(* CODESYS project DiagnosisEtherCAT.library
   Author: TK
   Version: 0.0.9.1
   Description: EtherCATのマスター、スレーブの診断用FBのライブラリです。
   Title: Tk_Diagnosis_EtherCAT
   Placeholder: Tk_Diagnosis_EtherCAT
   Company: Komatsu

Project tree, tasks and I/O mapping:
  libraries: Tc2_Standard, * (Beckhoff Automation GmbH); Tc2_System, * (Beckhoff Automation GmbH); Tc3_EventLogger, * (Beckhoff Automation GmbH)
  EtherCAT Master/
    Base/
      function block FB_DevStateDiagnosis [ST]: FB_Init
      function block FB_FrmStateDiagnosis [ST]: FB_Init
      function block FB_FrmWcStateDiagnosis [ST]: FB_Init
      function block FB_SlaveCountDiagnosis [ST]: FB_Init
    function block FB_DiagnosisEtherCATMaster [ST]
  EtherCAT Slave/
    Base/
      function block FB_StateDiagnosis [ST]: FB_Init
      function block FB_WcStateDiagnosis [ST]: FB_Init
    function block FB_DiagnosisEtherCATSlaveWc0 [ST]: bError, Execute
    function block FB_DiagnosisEtherCATSlaveWc1 [ST]: bError, Execute
    function block FB_DiagnosisEtherCATSlaveWc2 [ST]: bError, Execute
    interface I_DiagnosisEtherCATSlave: bError, Execute
  Example FB/
    function block FB_DiagnosisEtherCATExample [ST]: EtherCATMasterDiagnosis, EtherCATSlaveDiagnosis
  Version/
    global variables Global_Version
*)

// Version/Global_Version
{attribute 'TcGenerated'}
{attribute 'no-analysis'}
{attribute 'linkalways'}
// This function has been automatically generated from the project information.
VAR_GLOBAL CONSTANT
	{attribute 'const_non_replaced'}
	stLibVersion_Tk_Diagnosis_EtherCAT : ST_LibVersion := (iMajor := 0, iMinor := 0, iBuild := 9, iRevision := 1, nFlags := 0, sVersion := '0.0.9.1');
END_VAR

// EtherCAT Master/Base/FB_DevStateDiagnosis
FUNCTION_BLOCK FB_DevStateDiagnosis
VAR CONSTANT
	uiFaultMask					:UINT	:=2#0001_1111_1111_0011;	//デバイスエラーのマスク
END_VAR
VAR_INPUT
	sMasterName					:STRING	:='NameNotSet';				//マスター名
END_VAR
VAR_OUTPUT
	bError						:BOOL;								//エラー発生を出力
END_VAR
VAR
	uiDevState 			AT%I*	:UINT;								//PDデータとリンク
		
	bErrorState					:ARRAY[0..15] OF BOOL;				//各ステートエラー
	fbBitREdge					:ARRAY[0..15] OF R_TRIG;
	fbMessage					:ARRAY[0..15] OF FB_TcMessage;
	i							:INT;
END_VAR

//エラー状態を出力
	bError:= (uiDevState AND uiFaultMask)<>0 ;

//デバイスの状態チェック、エラーは複数発生する可能性があるので全bitチェック
	FOR i := 0 TO 15 DO
		bErrorState[i]:=(uiDevState AND SHL(1,i))<>0;
	END_FOR

//結果をEventloggerへ
	FOR i := 0 TO 15 BY 1 DO
		fbBitREdge[i](CLK:=bErrorState[i]);
		
		IF fbBitREdge[i].Q THEN
			fbMessage[i].ipArguments.Clear().AddString(sMasterName);
			fbMessage[i].Send();
		END_IF
		
	END_FOR

//FB_Init は常に暗黙的に使用可能で、主に初期化に使用されます。
//戻り値は評価されません。特定の結果を得るために、メソッドを明示的に宣言し、
//そのメソッドに標準の初期化コードをもったコードを追加することができます。戻り値を評価できます。
METHOD FB_Init: BOOL
VAR_INPUT
    bInitRetains: BOOL; // TRUE: 保持変数は初期化されます (ウォーム リセット、あるいはコールド リセット)
    bInCopyCode: BOOL;  // TRUE: 後でコードをコピーする (オンライン変更) ために、インスタンスをコピーします。
END_VAR
fbMessage[0].CreateEx(TC_EVENTS.TkEtherCATMasterDiagnosisEventClass.LinkError);
fbMessage[1].CreateEx(TC_EVENTS.TkEtherCATMasterDiagnosisEventClass.IOLockedAfterLinkErrorIOResetRequired);
fbMessage[2].CreateEx(TC_EVENTS.TkEtherCATMasterDiagnosisEventClass.LinkErrorRedundancyAdapter);
fbMessage[3].CreateEx(TC_EVENTS.TkEtherCATMasterDiagnosisEventClass.MissingOneFrameRedundancyAdapter);
fbMessage[4].CreateEx(TC_EVENTS.TkEtherCATMasterDiagnosisEventClass.OutOfSendResourcesIOResetRequired);
fbMessage[5].CreateEx(TC_EVENTS.TkEtherCATMasterDiagnosisEventClass.WatchdogTriggered);
fbMessage[6].CreateEx(TC_EVENTS.TkEtherCATMasterDiagnosisEventClass.EthernetDriverMiniportNotFound);
fbMessage[7].CreateEx(TC_EVENTS.TkEtherCATMasterDiagnosisEventClass.IOResetActive);
fbMessage[8].CreateEx(TC_EVENTS.TkEtherCATMasterDiagnosisEventClass.AtLeastOneDeviceInINITState);
fbMessage[9].CreateEx(TC_EVENTS.TkEtherCATMasterDiagnosisEventClass.AtLeastOneDeviceInPREOPState);
fbMessage[10].CreateEx(TC_EVENTS.TkEtherCATMasterDiagnosisEventClass.AtLeastOneDeviceInSAFEOPState);
fbMessage[11].CreateEx(TC_EVENTS.TkEtherCATMasterDiagnosisEventClass.AtLeastOneDeviceInERRORState);
fbMessage[12].CreateEx(TC_EVENTS.TkEtherCATMasterDiagnosisEventClass.DCNotInSync);
END_METHOD

END_FUNCTION_BLOCK

// EtherCAT Master/Base/FB_FrmStateDiagnosis
FUNCTION_BLOCK FB_FrmStateDiagnosis
VAR_INPUT
	sMasterName					:STRING	:='NameNotSet';				//マスター名
END_VAR
VAR_OUTPUT
	bError						:BOOL;								//エラー発生を出力
END_VAR
VAR
	uiFrmState 			AT%I*	:UINT;								//PDデータとリンク
	
	bErrorState					:ARRAY[0..15] OF BOOL;				//各ステートエラー
	fbBitREdge					:ARRAY[0..15] OF R_TRIG;
	bSendMsgMem					:ARRAY[0..14] OF BOOL;				//メッセージ送信を記憶	
	sSendMsgString				:STRING;							//送信メッセージのアーギュメント用
	bSendMsg					:BOOL;								//メッセージ送信予約
	fbMessage					:ARRAY[0..1] OF FB_TcMessage;
	i							:INT;
END_VAR

//エラー状態を出力
	bError:= uiFrmState<>0 ;
	
//サイクリックフレームごとのワーキングカウンターチェック、エラーは複数発生する可能性があるので全bitチェック
	FOR i := 0 TO 15 DO
		bErrorState[i]:=(uiFrmState AND SHL(1,i))<>0;
	END_FOR
	
//結果をEventloggerへ
	bSendMsg:=FALSE;	//メッセージ送信予約をリセット

	FOR i := 0 TO 14 BY 1 DO
		//エラーの立ち上がりエッジを検出
		fbBitREdge[i](CLK:=bErrorState[i]);
		
		//まだ送信していなければ、送信用の文字列作成
		IF NOT bSendMsgMem[i] AND fbBitREdge[i].Q THEN
			
			sSendMsgString:=CONCAT(sSendMsgString, CONCAT(INT_TO_STRING(i+1), '. '));	//送信メッセージのアーギュメント作成

			bSendMsg:=TRUE;		//メッセージ送信予約をセット
			bSendMsgMem[i]:=TRUE;	//メッセージ送信を記憶
			
		END_IF
		
		//エラーがリセットされたらメッセージ送信気を記憶をリセット
		IF NOT bErrorState[i] THEN
			bSendMsgMem[i]:=FALSE;
		END_IF
		
	END_FOR
	
	IF bSendMsg THEN
		fbMessage[0].ipArguments.Clear().AddString(sSendMsgString).AddString(sMasterName);
		fbMessage[0].Send();
		
		bSendMsg:=FALSE;
		sSendMsgString:='';
	END_IF
	
	//全体判定用
	fbBitREdge[15](CLK:=bErrorState[15]);
	
	IF fbBitREdge[15].Q THEN
		fbMessage[1].ipArguments.Clear().AddString(sMasterName);
		fbMessage[1].Send();
	END_IF

//FB_Init は常に暗黙的に使用可能で、主に初期化に使用されます。
//戻り値は評価されません。特定の結果を得るために、メソッドを明示的に宣言し、
//そのメソッドに標準の初期化コードをもったコードを追加することができます。戻り値を評価できます。
METHOD FB_Init: BOOL
VAR_INPUT
    bInitRetains: BOOL; // TRUE: 保持変数は初期化されます (ウォーム リセット、あるいはコールド リセット)
    bInCopyCode: BOOL;  // TRUE: 後でコードをコピーする (オンライン変更) ために、インスタンスをコピーします。
END_VAR
fbMessage[0].CreateEx(TC_EVENTS.TkEtherCATMasterDiagnosisEventClass.EtherCATCommandNotSentNOPRequested);
fbMessage[1].CreateEx(TC_EVENTS.TkEtherCATMasterDiagnosisEventClass.CompleteFrameNotSent);
END_METHOD

END_FUNCTION_BLOCK

// EtherCAT Master/Base/FB_FrmWcStateDiagnosis
FUNCTION_BLOCK FB_FrmWcStateDiagnosis
VAR_INPUT
	sMasterName					:STRING	:='NameNotSet';				//マスター名
END_VAR
VAR_OUTPUT
	bError						:BOOL;								//エラー発生を出力
END_VAR
VAR
	uiFrmWcState 		AT%I*	:UINT;								//PDデータとリンク
	
	bErrorState					:ARRAY[0..15] OF BOOL;				//各ステートエラー
	fbBitREdge					:ARRAY[0..15] OF R_TRIG;
	bSendMsgMem					:ARRAY[0..14] OF BOOL;				//メッセージ送信を記憶	
	sSendMsgString				:STRING;							//送信メッセージのアーギュメント用
	bSendMsg					:BOOL;								//メッセージ送信予約
	fbMessage					:ARRAY[0..1] OF FB_TcMessage;
	i							:INT;
END_VAR

//エラー状態を出力
	bError:= uiFrmWcState<>0 ;
	
//サイクリックフレームごとのワーキングカウンターチェック、エラーは複数発生する可能性があるので全bitチェック
	FOR i := 0 TO 15 DO
		bErrorState[i]:=(uiFrmWcState AND SHL(1,i))<>0;
	END_FOR
	
//結果をEventloggerへ
	bSendMsg:=FALSE;	//メッセージ送信予約をリセット

	FOR i := 0 TO 14 BY 1 DO
		//エラーの立ち上がりエッジを検出
		fbBitREdge[i](CLK:=bErrorState[i]);
		
		//まだ送信していなければ、送信用の文字列作成
		IF NOT bSendMsgMem[i] AND fbBitREdge[i].Q THEN
			
			sSendMsgString:=CONCAT(sSendMsgString, CONCAT(INT_TO_STRING(i+1), '. '));	//送信メッセージのアーギュメント作成

			bSendMsg:=TRUE;		//メッセージ送信予約をセット
			bSendMsgMem[i]:=TRUE;	//メッセージ送信を記憶
			
		END_IF
		
		//エラーがリセットされたらメッセージ送信気を記憶をリセット
		IF NOT bErrorState[i] THEN
			bSendMsgMem[i]:=FALSE;
		END_IF
		
	END_FOR
	
	IF bSendMsg THEN
		fbMessage[0].ipArguments.Clear().AddString(sSendMsgString).AddString(sMasterName);
		fbMessage[0].Send();
		
		bSendMsg:=FALSE;
		sSendMsgString:='';
	END_IF
	
	//全体判定用
	fbBitREdge[15](CLK:=bErrorState[15]);
	
	IF fbBitREdge[15].Q THEN
		fbMessage[1].ipArguments.Clear().AddString(sMasterName);
		fbMessage[1].Send();
	END_IF

//FB_Init は常に暗黙的に使用可能で、主に初期化に使用されます。
//戻り値は評価されません。特定の結果を得るために、メソッドを明示的に宣言し、
//そのメソッドに標準の初期化コードをもったコードを追加することができます。戻り値を評価できます。
METHOD FB_Init: BOOL
VAR_INPUT
    bInitRetains: BOOL; // TRUE: 保持変数は初期化されます (ウォーム リセット、あるいはコールド リセット)
    bInCopyCode: BOOL;  // TRUE: 後でコードをコピーする (オンライン変更) ために、インスタンスをコピーします。
END_VAR
fbMessage[0].CreateEx(TC_EVENTS.TkEtherCATMasterDiagnosisEventClass.WrongWorkingCounterEtherCATCommandReceived);
fbMessage[1].CreateEx(TC_EVENTS.TkEtherCATMasterDiagnosisEventClass.CompleteFrameMissing);
END_METHOD

END_FUNCTION_BLOCK

// EtherCAT Master/Base/FB_SlaveCountDiagnosis
FUNCTION_BLOCK FB_SlaveCountDiagnosis
VAR_INPUT
	sMasterName					:STRING	:='NameNotSet';				//マスター名
END_VAR
VAR_OUTPUT
	bError						:BOOL;								//エラー発生を出力
END_VAR
VAR
	uiSlaveCount 		AT%I*	:UINT;								//PDデータとリンク
	uiCfgSlaveCount 	AT%I*	:UINT;								//PDデータとリンク
	
	fbBitREdge					:R_TRIG;
	fbMessage					:FB_TcMessage;
	i							:INT;
END_VAR

//エラー状態を出力
	bError:=uiSlaveCount<>uiCfgSlaveCount OR uiSlaveCount=0 OR uiCfgSlaveCount=0;

//エラーをEventloggerへ
	fbBitREdge(CLK:=bError);
	
	IF fbBitREdge.Q THEN
		fbMessage.ipArguments.Clear().AddString(sMasterName);
		fbMessage.Send();
	END_IF

//FB_Init は常に暗黙的に使用可能で、主に初期化に使用されます。
//戻り値は評価されません。特定の結果を得るために、メソッドを明示的に宣言し、
//そのメソッドに標準の初期化コードをもったコードを追加することができます。戻り値を評価できます。
METHOD FB_Init: BOOL
VAR_INPUT
    bInitRetains: BOOL; // TRUE: 保持変数は初期化されます (ウォーム リセット、あるいはコールド リセット)
    bInCopyCode: BOOL;  // TRUE: 後でコードをコピーする (オンライン変更) ために、インスタンスをコピーします。
END_VAR
fbMessage.CreateEx(Tc_Events.TkEtherCATMasterDiagnosisEventClass.MismatchSlaveCountCfgSlaveCount);
END_METHOD

END_FUNCTION_BLOCK

// EtherCAT Master/FB_DiagnosisEtherCATMaster
FUNCTION_BLOCK FB_DiagnosisEtherCATMaster
VAR_INPUT
	sMasterName					:STRING	:='NameNotSet';				//マスター名
END_VAR
VAR_IN_OUT
	fbFrmWcStateDiagnosis		:ARRAY[*] OF FB_FrmWcStateDiagnosis;
	fbFrmStateDiagnosis			:ARRAY[*] OF FB_FrmStateDiagnosis;
END_VAR
VAR_OUTPUT
	bError						:BOOL;								//エラー発生を出力
END_VAR
VAR
	fbDevStateDiagnosis			:FB_DevStateDiagnosis;
	fbSlaveCountDiagnosis		:FB_SlaveCountDiagnosis;
	i							:DINT;
END_VAR

//診断用FBを呼び出し
fbDevStateDiagnosis(sMasterName:=sMasterName);
fbSlaveCountDiagnosis(sMasterName:=sMasterName);

bError:=fbDevStateDiagnosis.bError OR fbSlaveCountDiagnosis.bError;

//可変長のアレイを診断と出力
FOR i := LOWER_BOUND(fbFrmWcStateDiagnosis,1) TO UPPER_BOUND(fbFrmWcStateDiagnosis,1) DO
	fbFrmWcStateDiagnosis[i](sMasterName:=sMasterName);
	bError:=bError OR fbFrmWcStateDiagnosis[i].bError;
END_FOR

FOR i := LOWER_BOUND(fbFrmStateDiagnosis,1) TO UPPER_BOUND(fbFrmStateDiagnosis,1) DO
	fbFrmStateDiagnosis[i](sMasterName:=sMasterName);
	bError:=bError OR fbFrmStateDiagnosis[i].bError;
END_FOR

END_FUNCTION_BLOCK

// EtherCAT Slave/Base/FB_StateDiagnosis
FUNCTION_BLOCK FB_StateDiagnosis
VAR CONSTANT
	uiFaultMask					:UINT	:=2#1111_1111_1111_0111;	//デバイスエラーのマスク
END_VAR
VAR_INPUT
	sSlaveName					:STRING	:='NameNotSet';				//スレーブ名
END_VAR
VAR_OUTPUT
	bError						:BOOL;								//エラー発生を出力
END_VAR
VAR
	uiState				AT%I*	:UINT;								//PDデータとリンク
	
	bErrorState					:ARRAY[0..16] OF BOOL;				//各ステートエラー
	fbBitREdge					:ARRAY[0..16] OF R_TRIG;
	fbMessage					:ARRAY[0..16] OF FB_TcMessage;
	i							:INT;
END_VAR

//エラー状態を出力
	bError:= (uiState AND uiFaultMask)<>0 ;

//スレーブのステータスをbitから診断
	bErrorState[0]:=uiState.0 AND NOT uiState.1;
	bErrorState[1]:=uiState.1 AND NOT uiState.0;
	bErrorState[2]:=uiState.0 AND uiState.1;
	bErrorState[3]:=uiState.2;
	bErrorState[4]:=uiState.3;

//スレーブのエラーは複数発生する可能性があるので全bitチェック
	FOR i := 4 TO 15 DO
		bErrorState[i+1]:=(uiState AND SHL(1,i))<>0;
	END_FOR

//結果をEventloggerへ
	FOR i := 0 TO 16 BY 1 DO
		fbBitREdge[i](CLK:=bErrorState[i]);
		
		IF fbBitREdge[i].Q THEN
			fbMessage[i].ipArguments.Clear().AddString(sSlaveName);
			fbMessage[i].Send();
		END_IF
		
	END_FOR

//FB_Init は常に暗黙的に使用可能で、主に初期化に使用されます。
//戻り値は評価されません。特定の結果を得るために、メソッドを明示的に宣言し、
//そのメソッドに標準の初期化コードをもったコードを追加することができます。戻り値を評価できます。
METHOD FB_Init: BOOL
VAR_INPUT
    bInitRetains: BOOL; // TRUE: 保持変数は初期化されます (ウォーム リセット、あるいはコールド リセット)
    bInCopyCode: BOOL;  // TRUE: 後でコードをコピーする (オンライン変更) ために、インスタンスをコピーします。
END_VAR
fbMessage[0].CreateEx(TC_EVENTS.TkEtherCATSlaveDiagnosisEventClass.INIT);
fbMessage[1].CreateEx(TC_EVENTS.TkEtherCATSlaveDiagnosisEventClass.PREOP);
fbMessage[2].CreateEx(TC_EVENTS.TkEtherCATSlaveDiagnosisEventClass.BOOT);
fbMessage[3].CreateEx(TC_EVENTS.TkEtherCATSlaveDiagnosisEventClass.SAFEOP);
fbMessage[4].CreateEx(TC_EVENTS.TkEtherCATSlaveDiagnosisEventClass.OP);
fbMessage[5].CreateEx(TC_EVENTS.TkEtherCATSlaveDiagnosisEventClass.SlaveSignalsError);
fbMessage[6].CreateEx(TC_EVENTS.TkEtherCATSlaveDiagnosisEventClass.InvalidVendorIdProductCodeRead);
fbMessage[7].CreateEx(TC_EVENTS.TkEtherCATSlaveDiagnosisEventClass.InitializationErrorOccurred);
fbMessage[8].CreateEx(TC_EVENTS.TkEtherCATSlaveDiagnosisEventClass.SlaveDisabled);
fbMessage[9].CreateEx(TC_EVENTS.TkEtherCATSlaveDiagnosisEventClass.SlaveNotPresent);
fbMessage[10].CreateEx(TC_EVENTS.TkEtherCATSlaveDiagnosisEventClass.SlaveSignalsLinkError);
fbMessage[11].CreateEx(TC_EVENTS.TkEtherCATSlaveDiagnosisEventClass.SlaveSignalsMissingLink);
fbMessage[12].CreateEx(TC_EVENTS.TkEtherCATSlaveDiagnosisEventClass.SlaveSlaveSignalsUnexpectedLink);
fbMessage[13].CreateEx(TC_EVENTS.TkEtherCATSlaveDiagnosisEventClass.CommunicationPortA);
fbMessage[14].CreateEx(TC_EVENTS.TkEtherCATSlaveDiagnosisEventClass.CommunicationPortB);
fbMessage[15].CreateEx(TC_EVENTS.TkEtherCATSlaveDiagnosisEventClass.CommunicationPortC);
fbMessage[16].CreateEx(TC_EVENTS.TkEtherCATSlaveDiagnosisEventClass.CommunicationPortD);
END_METHOD

END_FUNCTION_BLOCK

// EtherCAT Slave/Base/FB_WcStateDiagnosis
FUNCTION_BLOCK FB_WcStateDiagnosis
VAR_INPUT
	sSlaveName					:STRING	:='NameNotSet';				//スレーブ名
END_VAR
VAR_OUTPUT
	bError						:BOOL;								//エラー発生を出力
END_VAR
VAR
	bWcState			AT%I*	:BOOL;								//PDデータとリンク
	
	fbBitREdge					:R_TRIG;
	fbMessage					:FB_TcMessage;
END_VAR

//エラー状態を出力
	bError:=bWcState;

//結果をEventloggerへ
	fbBitREdge(CLK:=bError);
	
	IF fbBitREdge.Q THEN
		fbMessage.ipArguments.Clear().AddString(sSlaveName);
		fbMessage.Send();
	END_IF

//FB_Init は常に暗黙的に使用可能で、主に初期化に使用されます。
//戻り値は評価されません。特定の結果を得るために、メソッドを明示的に宣言し、
//そのメソッドに標準の初期化コードをもったコードを追加することができます。戻り値を評価できます。
METHOD FB_Init: BOOL
VAR_INPUT
    bInitRetains: BOOL; // TRUE: 保持変数は初期化されます (ウォーム リセット、あるいはコールド リセット)
    bInCopyCode: BOOL;  // TRUE: 後でコードをコピーする (オンライン変更) ために、インスタンスをコピーします。
END_VAR
fbMessage.CreateEx(TC_EVENTS.TkEtherCATSlaveDiagnosisEventClass.InvalidWorkingCounter);
END_METHOD

END_FUNCTION_BLOCK

// EtherCAT Slave/FB_DiagnosisEtherCATSlaveWc0
FUNCTION_BLOCK FB_DiagnosisEtherCATSlaveWc0 IMPLEMENTS I_DiagnosisEtherCATSlave
VAR_INPUT
	sSlaveName					:STRING	:='NameNotSet';				//スレーブ名
END_VAR
VAR
	_bError						:BOOL;
	
	fbStateDiagnosis			:FB_StateDiagnosis;
END_VAR

(*エラー発生を出力*)
PROPERTY bError : BOOL
GET
bError:=_bError;
END_GET
END_PROPERTY

(*呼び出して診断実行*)
METHOD Execute
//診断用FBを呼び出し
fbStateDiagnosis(sSlaveName:=sSlaveName);

_bError:=fbStateDiagnosis.bError;
END_METHOD

END_FUNCTION_BLOCK

// EtherCAT Slave/I_DiagnosisEtherCATSlave
INTERFACE I_DiagnosisEtherCATSlave

//エラー発生を出力
PROPERTY bError : BOOL
GET
END_GET
END_PROPERTY

//呼び出して診断実行
METHOD Execute
VAR_INPUT
END_VAR
END_METHOD

END_INTERFACE

// EtherCAT Slave/FB_DiagnosisEtherCATSlaveWc1
FUNCTION_BLOCK FB_DiagnosisEtherCATSlaveWc1 IMPLEMENTS I_DiagnosisEtherCATSlave
VAR_INPUT
	sSlaveName					:STRING	:='NameNotSet';				//スレーブ名
END_VAR
VAR
	_bError						:BOOL;
	
	fbStateDiagnosis			:FB_StateDiagnosis;
	fbWcStateDiagnosis			:FB_WcStateDiagnosis;
END_VAR

(*エラー発生を出力*)
PROPERTY bError : BOOL
GET
bError:=_bError;
END_GET
END_PROPERTY

(*呼び出して診断実行*)
METHOD Execute
//診断用FBを呼び出し
fbStateDiagnosis(sSlaveName:=sSlaveName);
fbWcStateDiagnosis(sSlaveName:=sSlaveName);

_bError:=fbStateDiagnosis.bError OR fbWcStateDiagnosis.bError;
END_METHOD

END_FUNCTION_BLOCK

// EtherCAT Slave/FB_DiagnosisEtherCATSlaveWc2
FUNCTION_BLOCK FB_DiagnosisEtherCATSlaveWc2 IMPLEMENTS I_DiagnosisEtherCATSlave
VAR_INPUT
	sSlaveName					:STRING	:='NameNotSet';				//スレーブ名
END_VAR
VAR
	_bError						:BOOL;
	
	fbStateDiagnosis			:FB_StateDiagnosis;
	fbWcStateDiagnosis1			:FB_WcStateDiagnosis;
	fbWcStateDiagnosis2			:FB_WcStateDiagnosis;
END_VAR

(*エラー発生を出力*)
PROPERTY bError : BOOL
GET
bError:=_bError;
END_GET
END_PROPERTY

(*呼び出して診断実行*)
METHOD Execute
//診断用FBを呼び出し
fbStateDiagnosis(sSlaveName:=sSlaveName);
fbWcStateDiagnosis1(sSlaveName:=sSlaveName);
fbWcStateDiagnosis2(sSlaveName:=sSlaveName);

_bError:=fbStateDiagnosis.bError OR fbWcStateDiagnosis1.bError OR fbWcStateDiagnosis2.bError;
END_METHOD

END_FUNCTION_BLOCK

// Example FB/FB_DiagnosisEtherCATExample
FUNCTION_BLOCK FB_DiagnosisEtherCATExample
VAR_OUTPUT
	bError									:BOOL;																		//エラーを纏めて出力
END_VAR
VAR
	i										:DINT;																		//for loop用
	
	//デバイス3
	fbFrmWcStateDiagnosis3					:ARRAY[0..0] OF FB_FrmWcStateDiagnosis;										//EtherCAt Master3フレーム数のFB
	fbFrmStateDiagnosis3					:ARRAY[0..0] OF FB_FrmStateDiagnosis;										//EtherCAt Master3フレーム数のFB
	fbDiagnosisEtherCATMaster3				:FB_DiagnosisEtherCATMaster	:=(sMasterName:='Device3_EtherCAT');			//EtherCAt Master3診断用FB

	//EtherCATスレーブ
	fbTerm2									:FB_DiagnosisEtherCATSlaveWc1	:=(sSlaveName:='Term2_EL6224');				//EtherCAT Slave3診断用FB
	fbTerm3									:FB_DiagnosisEtherCATSlaveWc0	:=(sSlaveName:='Term3_EK1110');				//EtherCAT Slave3診断用FB
	fbTerm4									:FB_DiagnosisEtherCATSlaveWc1	:=(sSlaveName:='Term4_EK1828');				//EtherCAT Slave4診断用FB
	fbTerm5									:FB_DiagnosisEtherCATSlaveWc1	:=(sSlaveName:='Term5_EL3318');				//EtherCAT Slave5診断用FB
	
	
	aSlaveDiagnoses							:ARRAY[1..4] OF I_DiagnosisEtherCATSlave :=[fbTerm2,
																						fbTerm3,
																						fbTerm4,
																						fbTerm5];						//EtherCAT Slave診断実行用のインターフェース
	
END_VAR

bError:=EtherCATMasterDiagnosis() OR EtherCATSlaveDiagnosis();

METHOD PRIVATE EtherCATMasterDiagnosis : BOOL
	fbDiagnosisEtherCATMaster3(	fbFrmWcStateDiagnosis:=fbFrmWcStateDiagnosis3,
								fbFrmStateDiagnosis:=fbFrmStateDiagnosis3) ;
								
	EtherCATMasterDiagnosis:=fbDiagnosisEtherCATMaster3.bError;
END_METHOD

METHOD PRIVATE EtherCATSlaveDiagnosis : BOOL
	FOR i := LOWER_BOUND(aSlaveDiagnoses,1) TO UPPER_BOUND(aSlaveDiagnoses,1) DO
		aSlaveDiagnoses[i].Execute();
		EtherCATSlaveDiagnosis:=EtherCATSlaveDiagnosis OR aSlaveDiagnoses[i].bError;
	END_FOR
END_METHOD

END_FUNCTION_BLOCK
